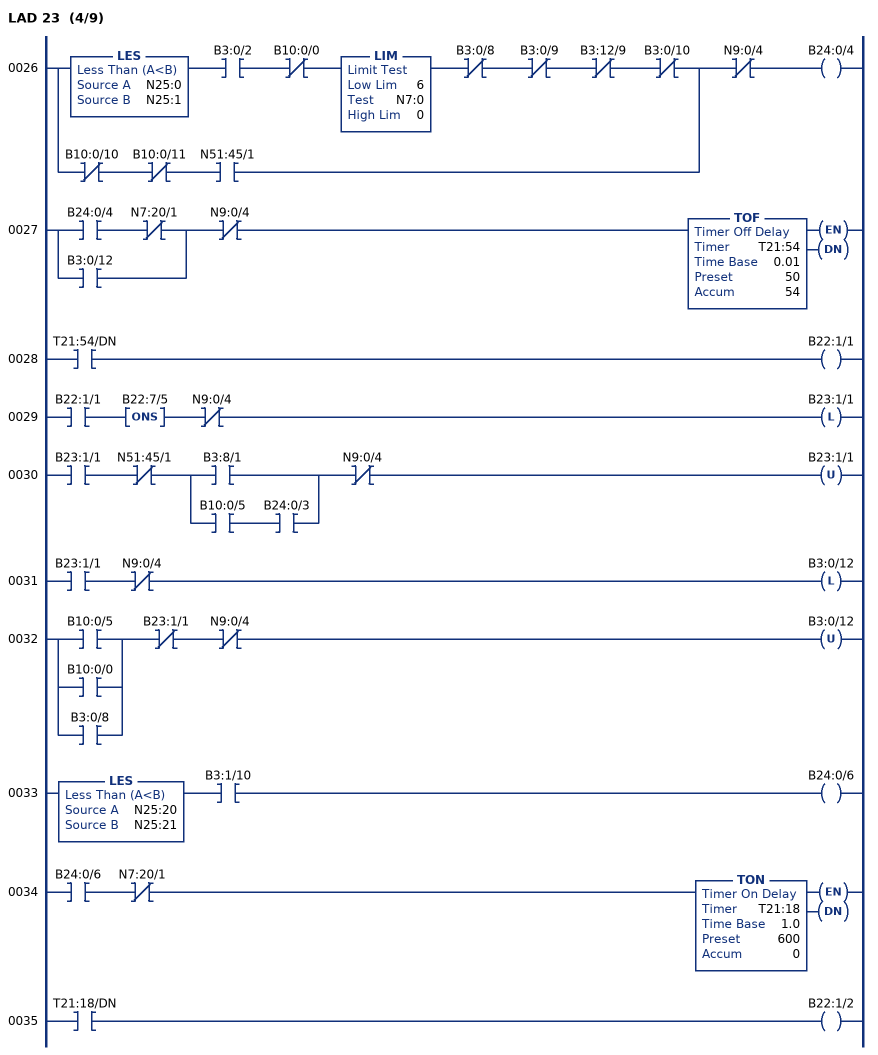
% Rung: 26 %
SOR BST LES N25:0 N25:1 XIC B3:0/2 XIO B10:0/0 LIM 6 N7:0 0 XIO B3:0/8 XIO B3:0/9 XIO B3:12/9 XIO B3:0/10 NXB XIO B10:0/10 XIO B10:0/11 XIC N51:45/1 BND XIO N9:0/4 OTE B24:0/4 EOR
% Rung: 27 %
SOR BST XIC B24:0/4 XIO N7:20/1 NXB XIC B3:0/12 BND XIO N9:0/4 TOF T21:54 0.01 50 54 EOR
% Rung: 28 %
SOR XIC T21:54/DN OTE B22:1/1 EOR
% Rung: 29 %
SOR XIC B22:1/1 OSR B22:7/5 XIO N9:0/4 OTL B23:1/1 EOR
% Rung: 30 %
SOR XIC B23:1/1 XIO N51:45/1 BST XIC B3:8/1 NXB XIC B10:0/5 XIC B24:0/3 BND XIO N9:0/4 OTU B23:1/1 EOR
% Rung: 31 %
SOR XIC B23:1/1 XIO N9:0/4 OTL B3:0/12 EOR
% Rung: 32 %
SOR BST XIC B10:0/5 NXB XIC B10:0/0 NXB XIC B3:0/8 BND XIO B23:1/1 XIO N9:0/4 OTU B3:0/12 EOR
% Rung: 33 %
SOR LES N25:20 N25:21 XIC B3:1/10 OTE B24:0/6 EOR
% Rung: 34 %
SOR XIC B24:0/6 XIO N7:20/1 TON T21:18 1.0 600 0 EOR
% Rung: 35 %
SOR XIC T21:18/DN OTE B22:1/2 EOR

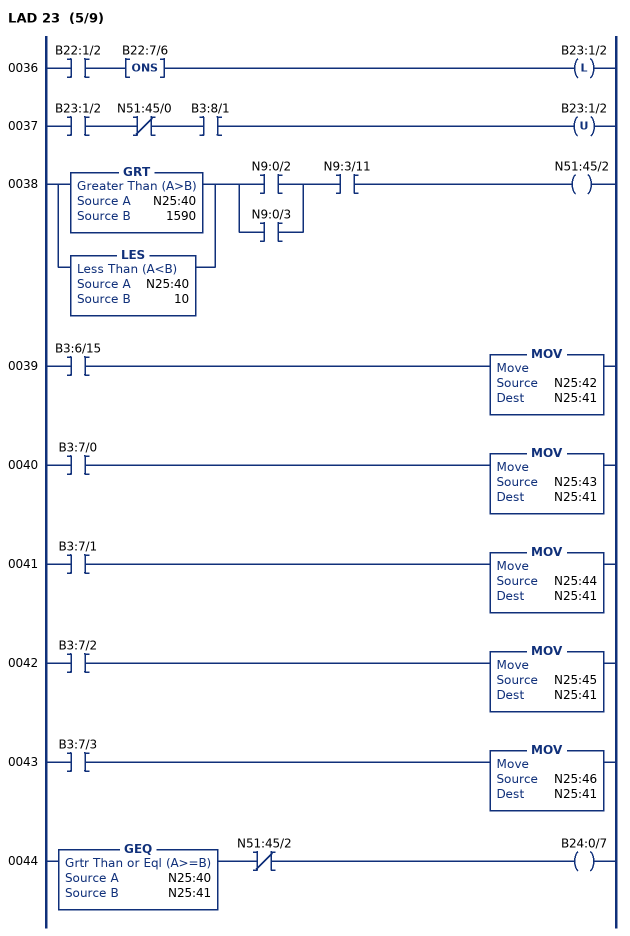
% Rung: 36 %
SOR XIC B22:1/2 OSR B22:7/6 OTL B23:1/2 EOR
% Rung: 37 %
SOR XIC B23:1/2 XIO N51:45/0 XIC B3:8/1 OTU B23:1/2 EOR
% Rung: 38 %
SOR BST GRT N25:40 1590 NXB LES N25:40 10 BND BST XIC N9:0/2 NXB XIC N9:0/3 BND XIC N9:3/11 OTE N51:45/2 EOR
% Rung: 39 %
SOR XIC B3:6/15 MOV N25:42 N25:41 EOR
% Rung: 40 %
SOR XIC B3:7/0 MOV N25:43 N25:41 EOR
% Rung: 41 %
SOR XIC B3:7/1 MOV N25:44 N25:41 EOR
% Rung: 42 %
SOR XIC B3:7/2 MOV N25:45 N25:41 EOR
% Rung: 43 %
SOR XIC B3:7/3 MOV N25:46 N25:41 EOR
% Rung: 44 %
SOR GEQ N25:40 N25:41 XIO N51:45/2 OTE B24:0/7 EOR

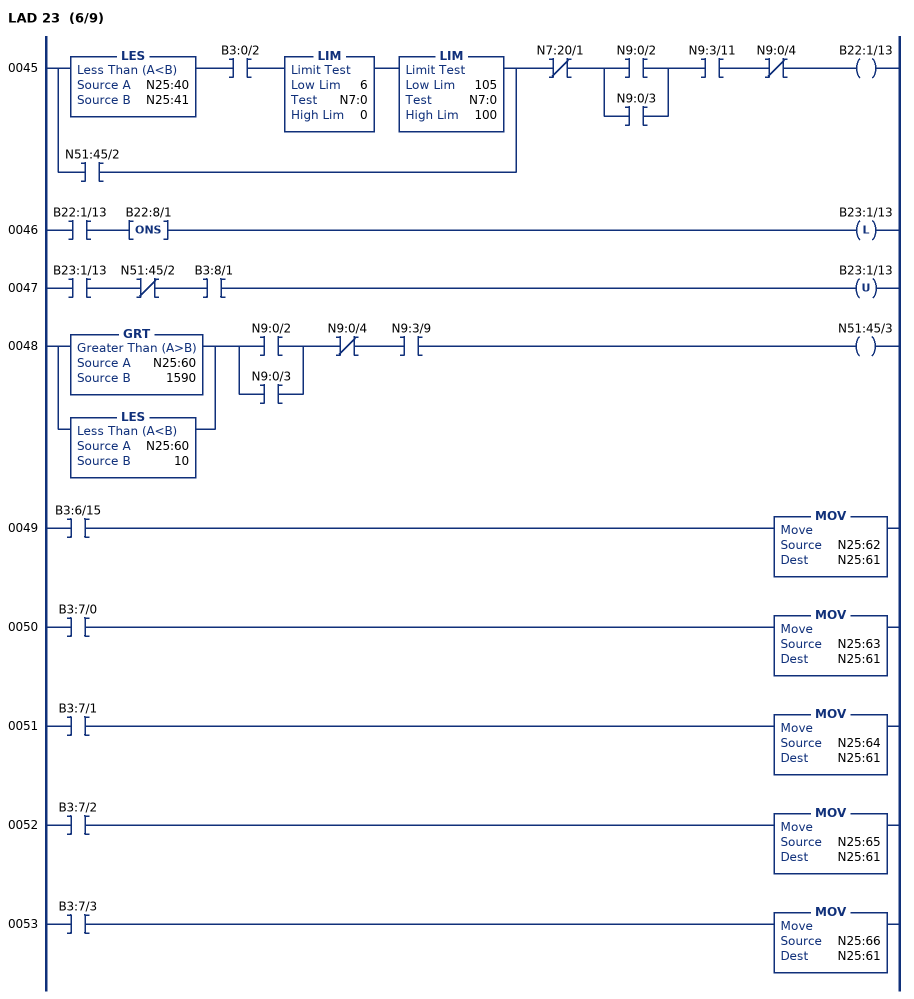
% Rung: 45 %
SOR BST LES N25:40 N25:41 XIC B3:0/2 LIM 6 N7:0 0 LIM 105 N7:0 100 NXB XIC N51:45/2 BND XIO N7:20/1 BST XIC N9:0/2 NXB XIC N9:0/3 BND XIC N9:3/11 XIO N9:0/4 OTE B22:1/13 EOR
% Rung: 46 %
SOR XIC B22:1/13 OSR B22:8/1 OTL B23:1/13 EOR
% Rung: 47 %
SOR XIC B23:1/13 XIO N51:45/2 XIC B3:8/1 OTU B23:1/13 EOR
% Rung: 48 %
SOR BST GRT N25:60 1590 NXB LES N25:60 10 BND BST XIC N9:0/2 NXB XIC N9:0/3 BND XIO N9:0/4 XIC N9:3/9 OTE N51:45/3 EOR
% Rung: 49 %
SOR XIC B3:6/15 MOV N25:62 N25:61 EOR
% Rung: 50 %
SOR XIC B3:7/0 MOV N25:63 N25:61 EOR
% Rung: 51 %
SOR XIC B3:7/1 MOV N25:64 N25:61 EOR
% Rung: 52 %
SOR XIC B3:7/2 MOV N25:65 N25:61 EOR
% Rung: 53 %
SOR XIC B3:7/3 MOV N25:66 N25:61 EOR

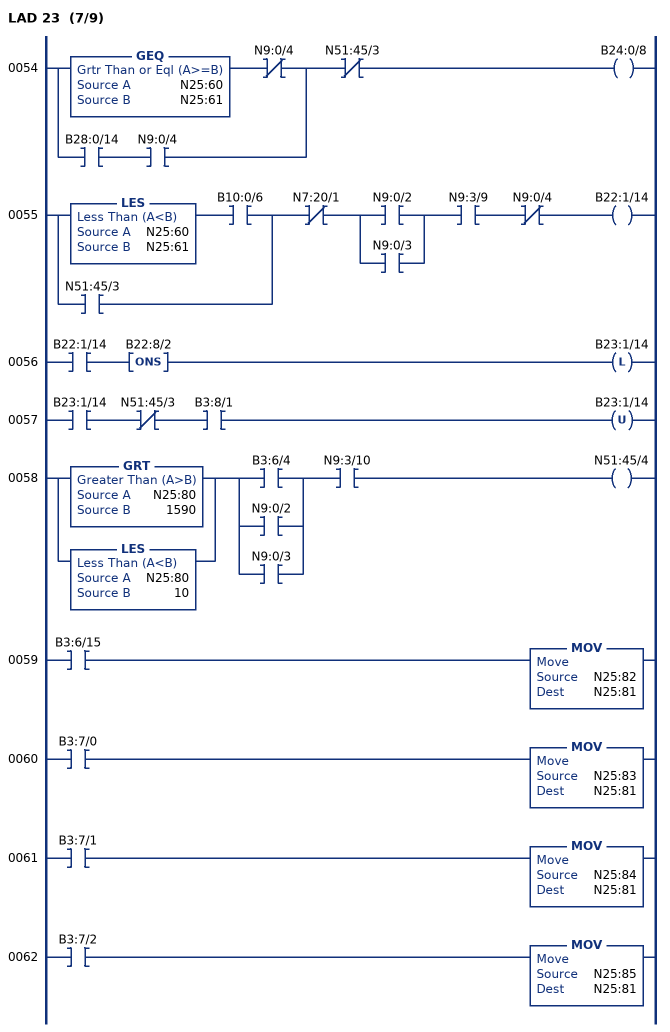
% Rung: 54 %
SOR BST GEQ N25:60 N25:61 XIO N9:0/4 NXB XIC B28:0/14 XIC N9:0/4 BND XIO N51:45/3 OTE B24:0/8 EOR
% Rung: 55 %
SOR BST LES N25:60 N25:61 XIC B10:0/6 NXB XIC N51:45/3 BND XIO N7:20/1 BST XIC N9:0/2 NXB XIC N9:0/3 BND XIC N9:3/9 XIO N9:0/4 OTE B22:1/14 EOR
% Rung: 56 %
SOR XIC B22:1/14 OSR B22:8/2 OTL B23:1/14 EOR
% Rung: 57 %
SOR XIC B23:1/14 XIO N51:45/3 XIC B3:8/1 OTU B23:1/14 EOR
% Rung: 58 %
SOR BST GRT N25:80 1590 NXB LES N25:80 10 BND BST XIC B3:6/4 NXB XIC N9:0/2 NXB XIC N9:0/3 BND XIC N9:3/10 OTE N51:45/4 EOR
% Rung: 59 %
SOR XIC B3:6/15 MOV N25:82 N25:81 EOR
% Rung: 60 %
SOR XIC B3:7/0 MOV N25:83 N25:81 EOR
% Rung: 61 %
SOR XIC B3:7/1 MOV N25:84 N25:81 EOR
% Rung: 62 %
SOR XIC B3:7/2 MOV N25:85 N25:81 EOR

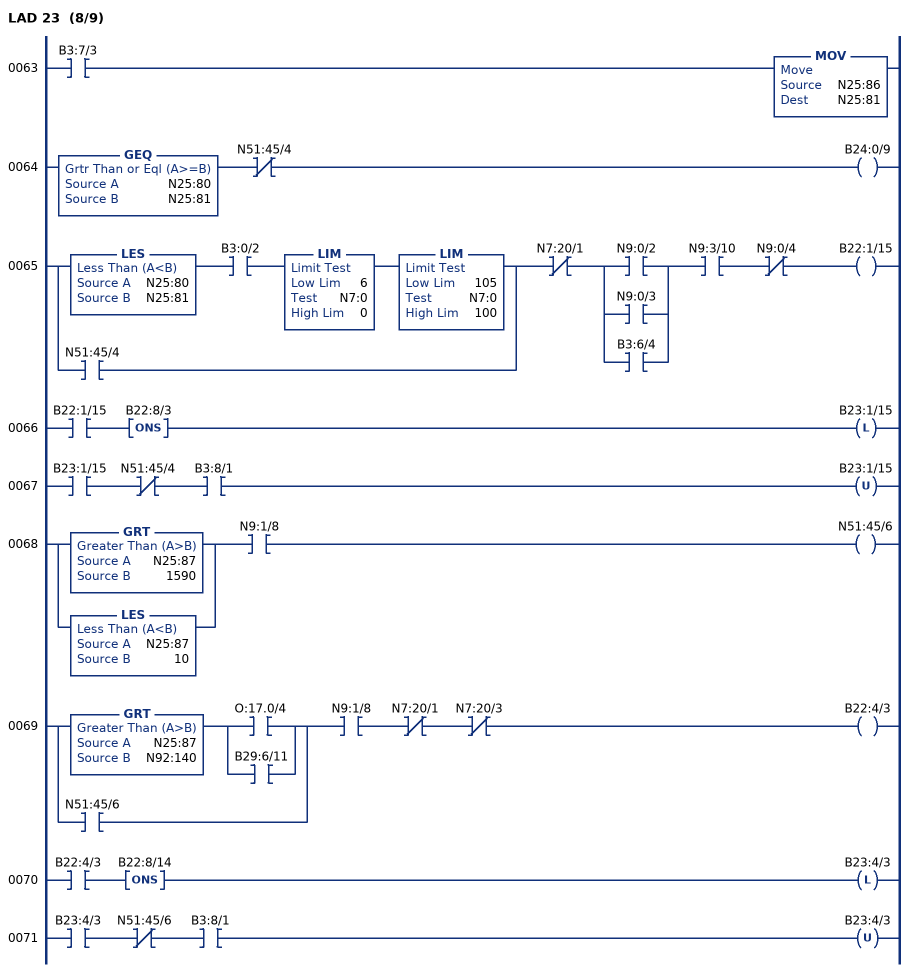
% Rung: 63 %
SOR XIC B3:7/3 MOV N25:86 N25:81 EOR
% Rung: 64 %
SOR GEQ N25:80 N25:81 XIO N51:45/4 OTE B24:0/9 EOR
% Rung: 65 %
SOR BST LES N25:80 N25:81 XIC B3:0/2 LIM 6 N7:0 0 LIM 105 N7:0 100 NXB XIC N51:45/4 BND XIO N7:20/1 BST XIC N9:0/2 NXB XIC N9:0/3 NXB XIC B3:6/4 BND XIC N9:3/10 XIO N9:0/4 OTE B22:1/15 EOR
% Rung: 66 %
SOR XIC B22:1/15 OSR B22:8/3 OTL B23:1/15 EOR
% Rung: 67 %
SOR XIC B23:1/15 XIO N51:45/4 XIC B3:8/1 OTU B23:1/15 EOR
% Rung: 68 %
SOR BST GRT N25:87 1590 NXB LES N25:87 10 BND XIC N9:1/8 OTE N51:45/6 EOR
% Rung: 69 %
SOR BST GRT N25:87 N92:140 BST XIC O:17.0/4 NXB XIC B29:6/11 BND NXB XIC N51:45/6 BND XIC N9:1/8 XIO N7:20/1 XIO N7:20/3 OTE B22:4/3 EOR
% Rung: 70 %
SOR XIC B22:4/3 OSR B22:8/14 OTL B23:4/3 EOR
% Rung: 71 %
SOR XIC B23:4/3 XIO N51:45/6 XIC B3:8/1 OTU B23:4/3 EOR

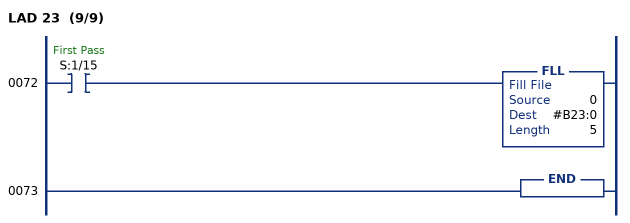
% Rung: 72 %
SOR XIC S:1/15 FLL 0 #B23:0 5 EOR
%   S:1/15  "First Pass" %
% Rung: 73 %
SOR END EOR

LADDER 24
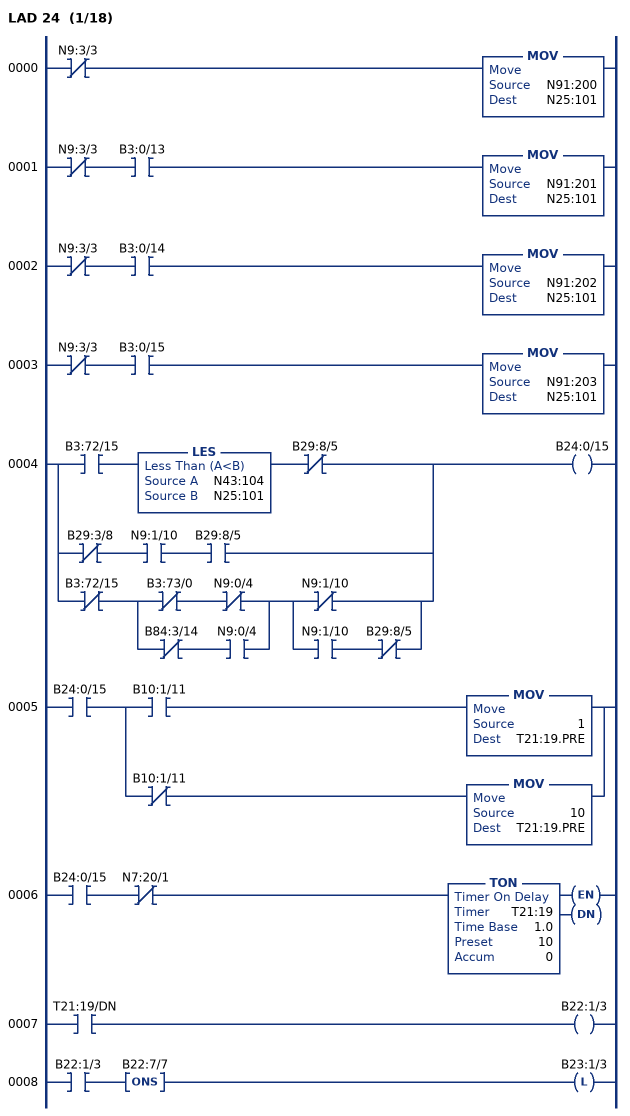
% Rung: 0 %
SOR XIO N9:3/3 MOV N91:200 N25:101 EOR
% Rung: 1 %
SOR XIO N9:3/3 XIC B3:0/13 MOV N91:201 N25:101 EOR
% Rung: 2 %
SOR XIO N9:3/3 XIC B3:0/14 MOV N91:202 N25:101 EOR
% Rung: 3 %
SOR XIO N9:3/3 XIC B3:0/15 MOV N91:203 N25:101 EOR
% Rung: 4 %
SOR BST XIC B3:72/15 LES N43:104 N25:101 XIO B29:8/5 NXB XIO B29:3/8 XIC N9:1/10 XIC B29:8/5 NXB XIO B3:72/15 BST XIO B3:73/0 XIO N9:0/4 NXB XIO B84:3/14 XIC N9:0/4 BND BST XIO N9:1/10 NXB XIC N9:1/10 XIO B29:8/5 BND BND OTE B24:0/15 EOR
% Rung: 5 %
SOR XIC B24:0/15 BST XIC B10:1/11 MOV 1 T21:19.PRE NXB XIO B10:1/11 MOV 10 T21:19.PRE BND EOR
% Rung: 6 %
SOR XIC B24:0/15 XIO N7:20/1 TON T21:19 1.0 10 0 EOR
% Rung: 7 %
SOR XIC T21:19/DN OTE B22:1/3 EOR
% Rung: 8 %
SOR XIC B22:1/3 OSR B22:7/7 OTL B23:1/3 EOR

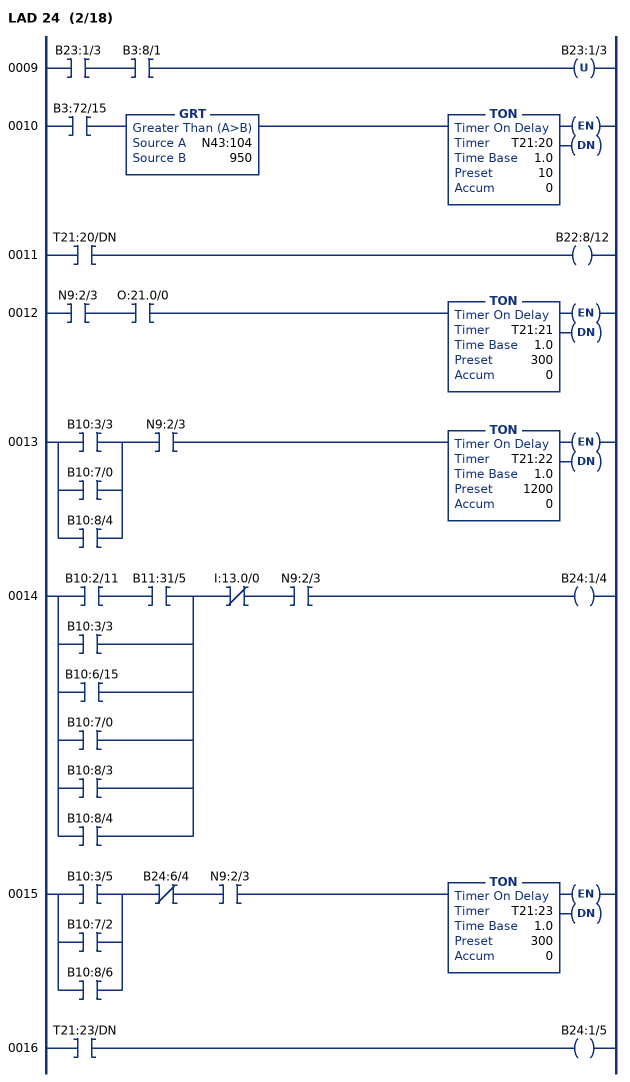
% Rung: 9 %
SOR XIC B23:1/3 XIC B3:8/1 OTU B23:1/3 EOR
% Rung: 10 %
SOR XIC B3:72/15 GRT N43:104 950 TON T21:20 1.0 10 0 EOR
% Rung: 11 %
SOR XIC T21:20/DN OTE B22:8/12 EOR
% Rung: 12 %
SOR XIC N9:2/3 XIC O:21.0/0 TON T21:21 1.0 300 0 EOR
% Rung: 13 %
SOR BST XIC B10:3/3 NXB XIC B10:7/0 NXB XIC B10:8/4 BND XIC N9:2/3 TON T21:22 1.0 1200 0 EOR
% Rung: 14 %
SOR BST XIC B10:2/11 XIC B11:31/5 NXB XIC B10:3/3 NXB XIC B10:6/15 NXB XIC B10:7/0 NXB XIC B10:8/3 NXB XIC B10:8/4 BND XIO I:13.0/0 XIC N9:2/3 OTE B24:1/4 EOR
% Rung: 15 %
SOR BST XIC B10:3/5 NXB XIC B10:7/2 NXB XIC B10:8/6 BND XIO B24:6/4 XIC N9:2/3 TON T21:23 1.0 300 0 EOR
% Rung: 16 %
SOR XIC T21:23/DN OTE B24:1/5 EOR

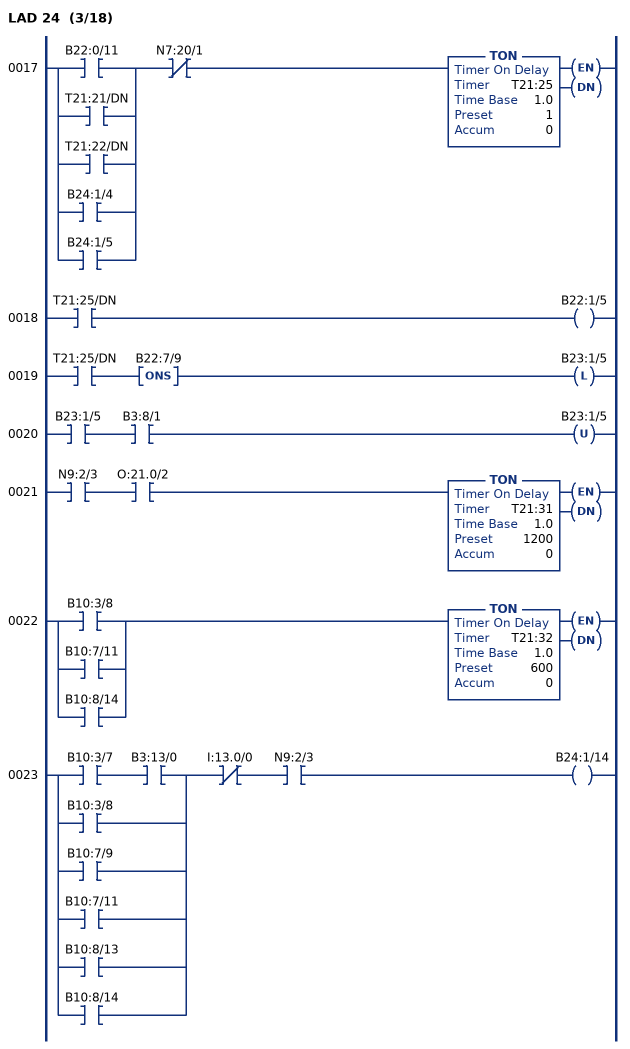
% Rung: 17 %
SOR BST XIC B22:0/11 NXB XIC T21:21/DN NXB XIC T21:22/DN NXB XIC B24:1/4 NXB XIC B24:1/5 BND XIO N7:20/1 TON T21:25 1.0 1 0 EOR
% Rung: 18 %
SOR XIC T21:25/DN OTE B22:1/5 EOR
% Rung: 19 %
SOR XIC T21:25/DN OSR B22:7/9 OTL B23:1/5 EOR
% Rung: 20 %
SOR XIC B23:1/5 XIC B3:8/1 OTU B23:1/5 EOR
% Rung: 21 %
SOR XIC N9:2/3 XIC O:21.0/2 TON T21:31 1.0 1200 0 EOR
% Rung: 22 %
SOR BST XIC B10:3/8 NXB XIC B10:7/11 NXB XIC B10:8/14 BND TON T21:32 1.0 600 0 EOR
% Rung: 23 %
SOR BST XIC B10:3/7 XIC B3:13/0 NXB XIC B10:3/8 NXB XIC B10:7/9 NXB XIC B10:7/11 NXB XIC B10:8/13 NXB XIC B10:8/14 BND XIO I:13.0/0 XIC N9:2/3 OTE B24:1/14 EOR

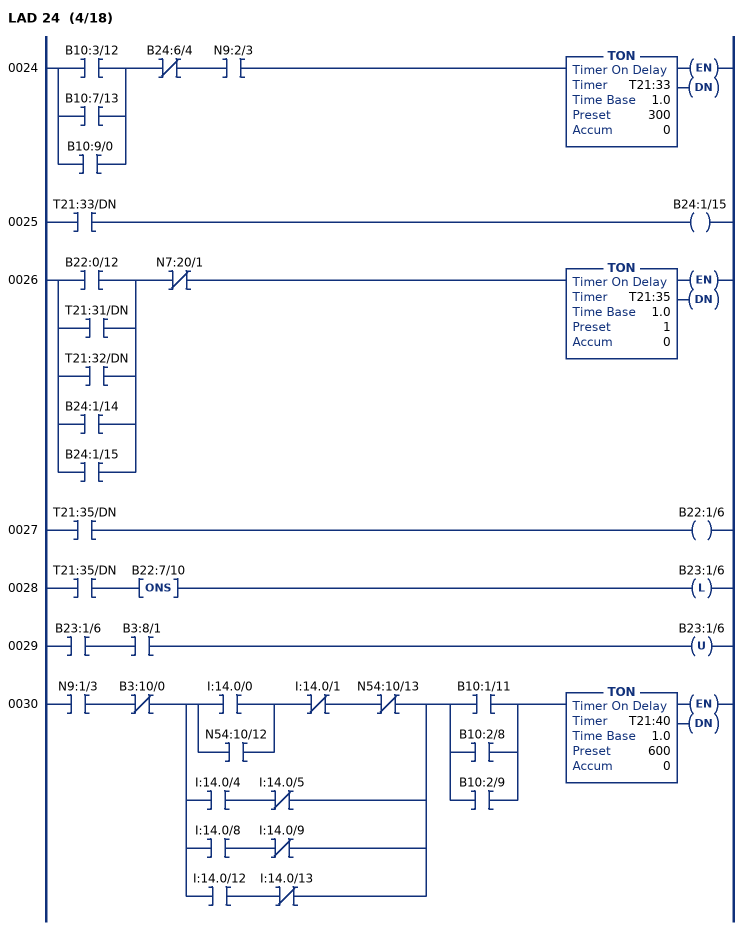
% Rung: 24 %
SOR BST XIC B10:3/12 NXB XIC B10:7/13 NXB XIC B10:9/0 BND XIO B24:6/4 XIC N9:2/3 TON T21:33 1.0 300 0 EOR
% Rung: 25 %
SOR XIC T21:33/DN OTE B24:1/15 EOR
% Rung: 26 %
SOR BST XIC B22:0/12 NXB XIC T21:31/DN NXB XIC T21:32/DN NXB XIC B24:1/14 NXB XIC B24:1/15 BND XIO N7:20/1 TON T21:35 1.0 1 0 EOR
% Rung: 27 %
SOR XIC T21:35/DN OTE B22:1/6 EOR
% Rung: 28 %
SOR XIC T21:35/DN OSR B22:7/10 OTL B23:1/6 EOR
% Rung: 29 %
SOR XIC B23:1/6 XIC B3:8/1 OTU B23:1/6 EOR
% Rung: 30 %
SOR XIC N9:1/3 XIO B3:10/0 BST BST XIC I:14.0/0 NXB XIC N54:10/12 BND XIO I:14.0/1 XIO N54:10/13 NXB XIC I:14.0/4 XIO I:14.0/5 NXB XIC I:14.0/8 XIO I:14.0/9 NXB XIC I:14.0/12 XIO I:14.0/13 BND BST XIC B10:1/11 NXB XIC B10:2/8 NXB XIC B10:2/9 BND TON T21:40 1.0 600 0 EOR

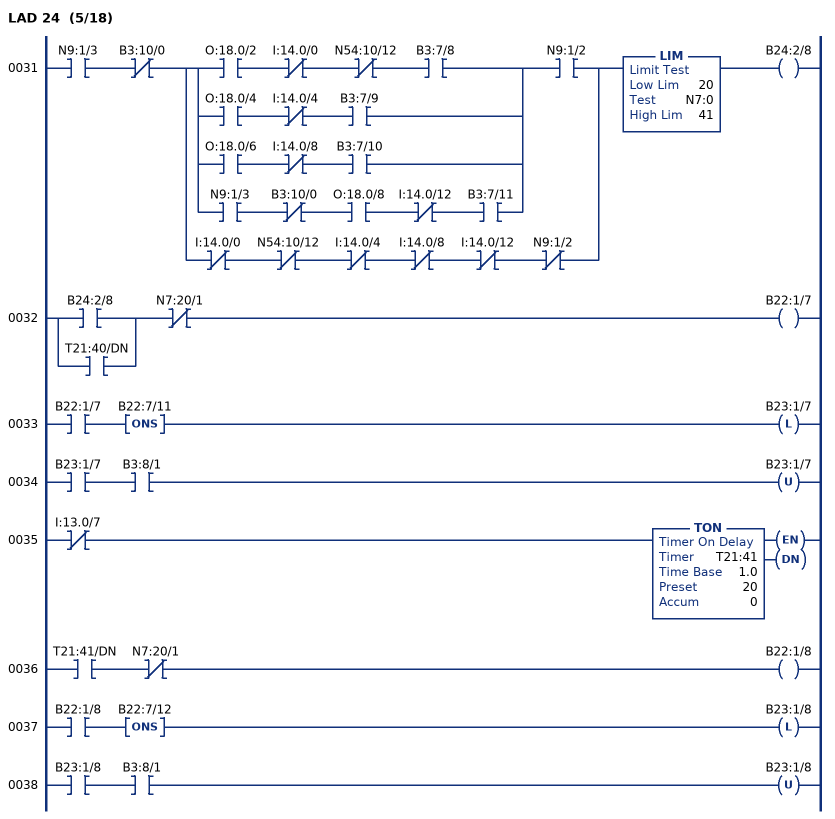
% Rung: 31 %
SOR XIC N9:1/3 XIO B3:10/0 BST BST XIC O:18.0/2 XIO I:14.0/0 XIO N54:10/12 XIC B3:7/8 NXB XIC O:18.0/4 XIO I:14.0/4 XIC B3:7/9 NXB XIC O:18.0/6 XIO I:14.0/8 XIC B3:7/10 NXB XIC N9:1/3 XIO B3:10/0 XIC O:18.0/8 XIO I:14.0/12 XIC B3:7/11 BND XIC N9:1/2 NXB XIO I:14.0/0 XIO N54:10/12 XIO I:14.0/4 XIO I:14.0/8 XIO I:14.0/12 XIO N9:1/2 BND LIM 20 N7:0 41 OTE B24:2/8 EOR
% Rung: 32 %
SOR BST XIC B24:2/8 NXB XIC T21:40/DN BND XIO N7:20/1 OTE B22:1/7 EOR
% Rung: 33 %
SOR XIC B22:1/7 OSR B22:7/11 OTL B23:1/7 EOR
% Rung: 34 %
SOR XIC B23:1/7 XIC B3:8/1 OTU B23:1/7 EOR
% Rung: 35 %
SOR XIO I:13.0/7 TON T21:41 1.0 20 0 EOR
% Rung: 36 %
SOR XIC T21:41/DN XIO N7:20/1 OTE B22:1/8 EOR
% Rung: 37 %
SOR XIC B22:1/8 OSR B22:7/12 OTL B23:1/8 EOR
% Rung: 38 %
SOR XIC B23:1/8 XIC B3:8/1 OTU B23:1/8 EOR

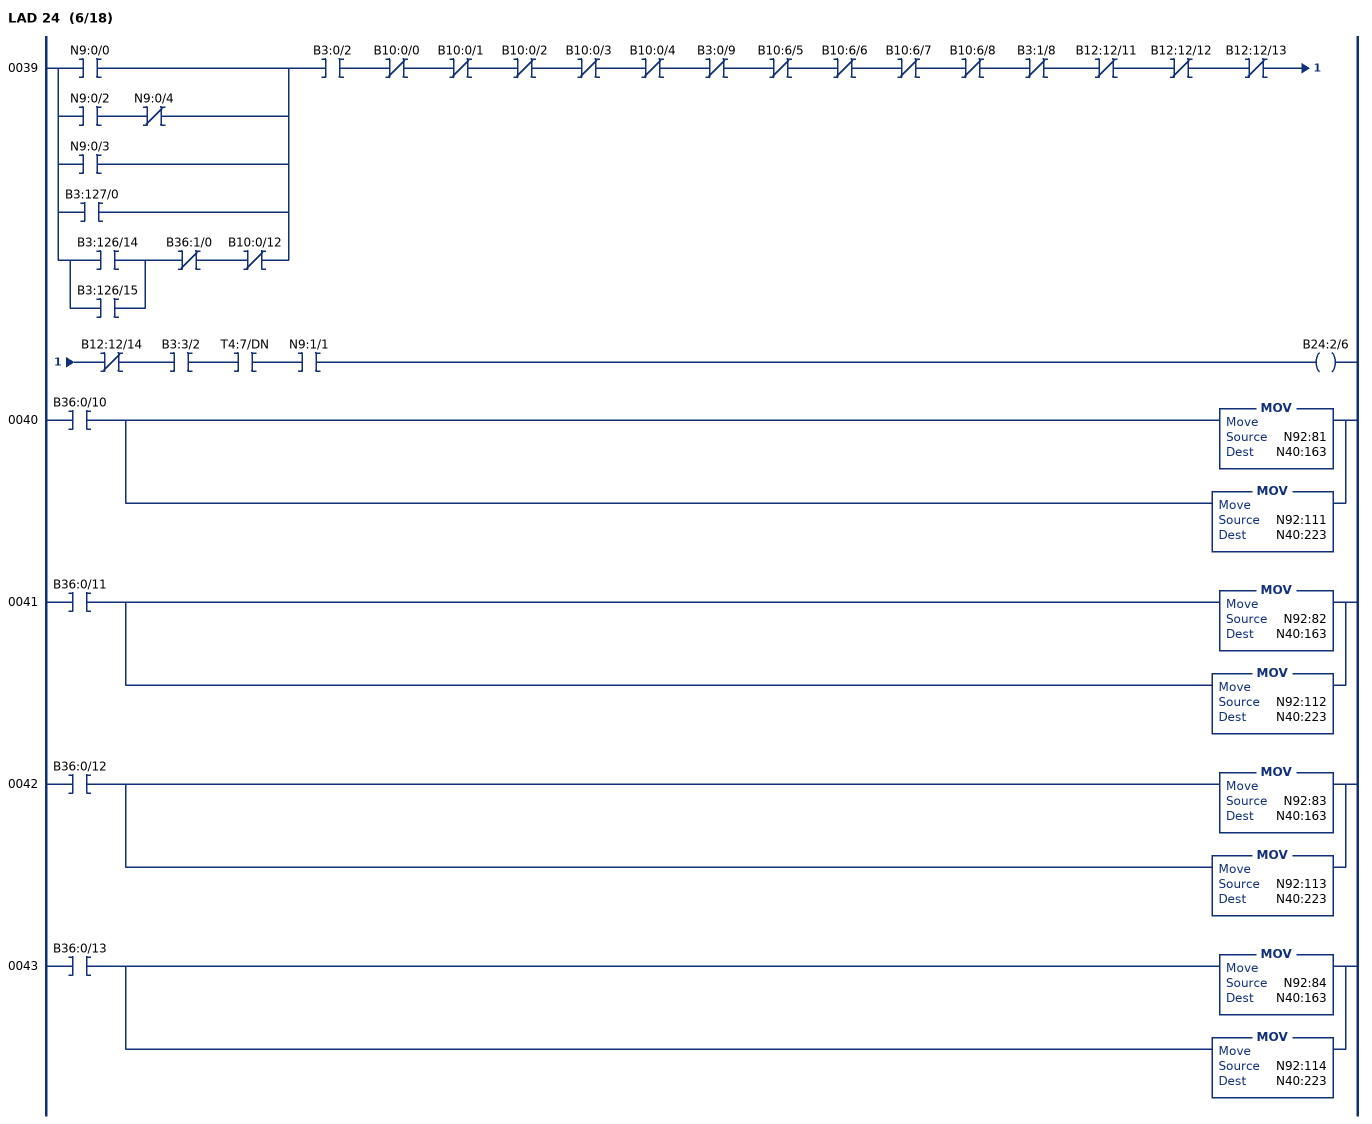
% Rung: 39 %
SOR BST XIC N9:0/0 NXB XIC N9:0/2 XIO N9:0/4 NXB XIC N9:0/3 NXB XIC B3:127/0 NXB BST XIC B3:126/14 NXB XIC B3:126/15 BND XIO B36:1/0 XIO B10:0/12 BND XIC B3:0/2 XIO B10:0/0 XIO B10:0/1 XIO B10:0/2 XIO B10:0/3 XIO B10:0/4 XIO B3:0/9 XIO B10:6/5 XIO B10:6/6 XIO B10:6/7 XIO B10:6/8 XIO B3:1/8 XIO B12:12/11 XIO B12:12/12 XIO B12:12/13 XIO B12:12/14 XIC B3:3/2 XIC T4:7/DN XIC N9:1/1 OTE B24:2/6 EOR
% Rung: 40 %
SOR XIC B36:0/10 BST MOV N92:81 N40:163 NXB MOV N92:111 N40:223 BND EOR
% Rung: 41 %
SOR XIC B36:0/11 BST MOV N92:82 N40:163 NXB MOV N92:112 N40:223 BND EOR
% Rung: 42 %
SOR XIC B36:0/12 BST MOV N92:83 N40:163 NXB MOV N92:113 N40:223 BND EOR
% Rung: 43 %
SOR XIC B36:0/13 BST MOV N92:84 N40:163 NXB MOV N92:114 N40:223 BND EOR

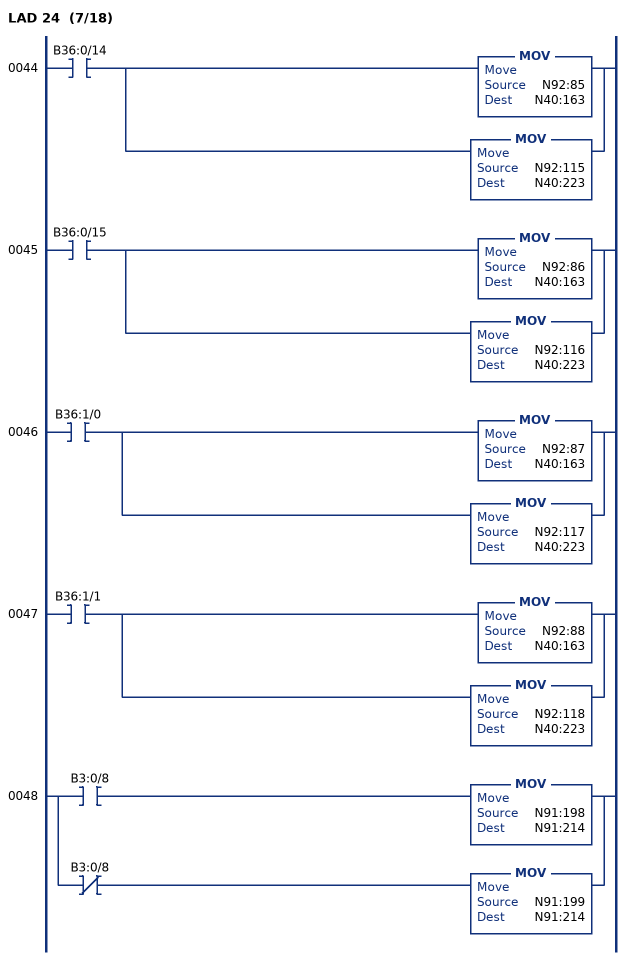
% Rung: 44 %
SOR XIC B36:0/14 BST MOV N92:85 N40:163 NXB MOV N92:115 N40:223 BND EOR
% Rung: 45 %
SOR XIC B36:0/15 BST MOV N92:86 N40:163 NXB MOV N92:116 N40:223 BND EOR
% Rung: 46 %
SOR XIC B36:1/0 BST MOV N92:87 N40:163 NXB MOV N92:117 N40:223 BND EOR
% Rung: 47 %
SOR XIC B36:1/1 BST MOV N92:88 N40:163 NXB MOV N92:118 N40:223 BND EOR
% Rung: 48 %
SOR BST XIC B3:0/8 MOV N91:198 N91:214 NXB XIO B3:0/8 MOV N91:199 N91:214 BND EOR

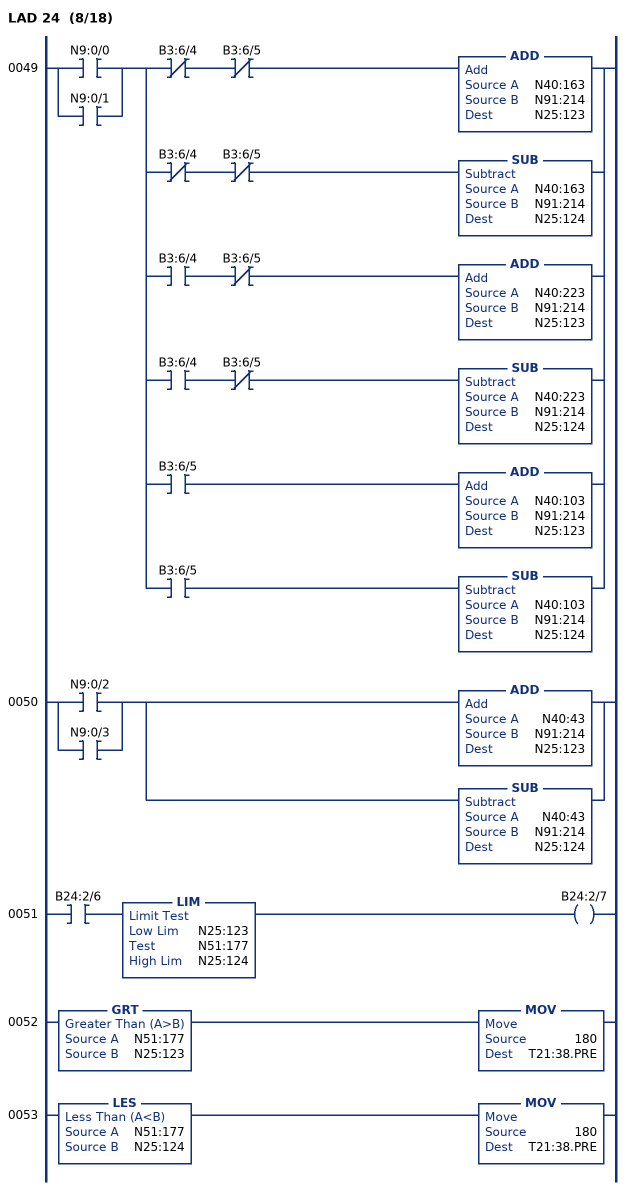
% Rung: 49 %
SOR BST XIC N9:0/0 NXB XIC N9:0/1 BND BST XIO B3:6/4 XIO B3:6/5 ADD N40:163 N91:214 N25:123 NXB XIO B3:6/4 XIO B3:6/5 SUB N40:163 N91:214 N25:124 NXB XIC B3:6/4 XIO B3:6/5 ADD N40:223 N91:214 N25:123 NXB XIC B3:6/4 XIO B3:6/5 SUB N40:223 N91:214 N25:124 NXB XIC B3:6/5 ADD N40:103 N91:214 N25:123 NXB XIC B3:6/5 SUB N40:103 N91:214 N25:124 BND EOR
% Rung: 50 %
SOR BST XIC N9:0/2 NXB XIC N9:0/3 BND BST ADD N40:43 N91:214 N25:123 NXB SUB N40:43 N91:214 N25:124 BND EOR
% Rung: 51 %
SOR XIC B24:2/6 LIM N25:123 N51:177 N25:124 OTE B24:2/7 EOR
% Rung: 52 %
SOR GRT N51:177 N25:123 MOV 180 T21:38.PRE EOR
% Rung: 53 %
SOR LES N51:177 N25:124 MOV 180 T21:38.PRE EOR

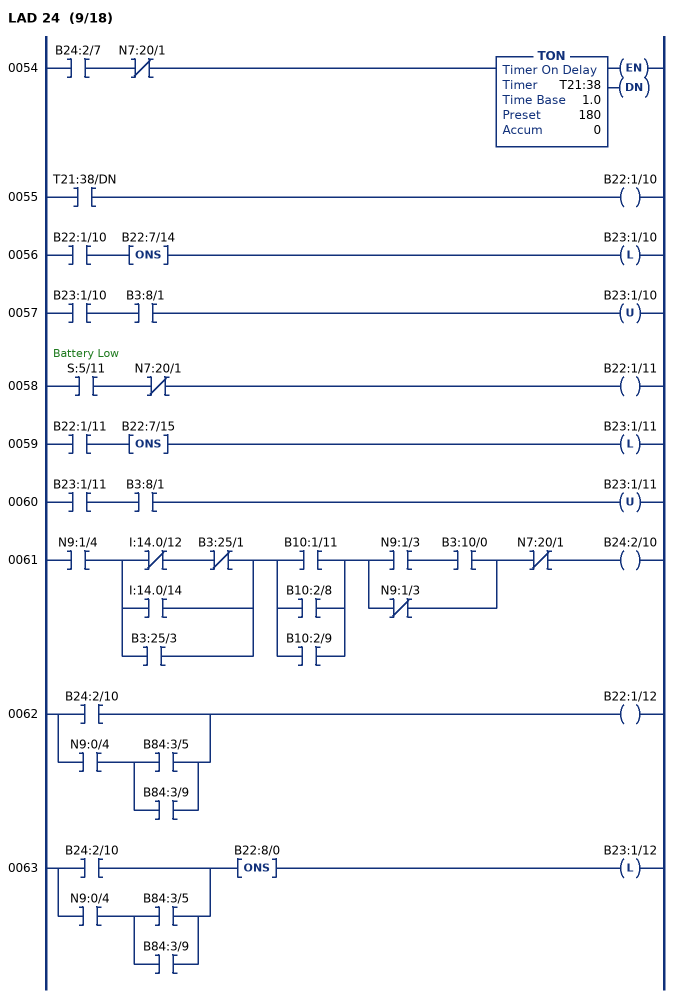
% Rung: 54 %
SOR XIC B24:2/7 XIO N7:20/1 TON T21:38 1.0 180 0 EOR
% Rung: 55 %
SOR XIC T21:38/DN OTE B22:1/10 EOR
% Rung: 56 %
SOR XIC B22:1/10 OSR B22:7/14 OTL B23:1/10 EOR
% Rung: 57 %
SOR XIC B23:1/10 XIC B3:8/1 OTU B23:1/10 EOR
% Rung: 58 %
SOR XIC S:5/11 XIO N7:20/1 OTE B22:1/11 EOR
%   S:5/11  "Battery Low" %
% Rung: 59 %
SOR XIC B22:1/11 OSR B22:7/15 OTL B23:1/11 EOR
% Rung: 60 %
SOR XIC B23:1/11 XIC B3:8/1 OTU B23:1/11 EOR
% Rung: 61 %
SOR XIC N9:1/4 BST XIO I:14.0/12 XIO B3:25/1 NXB XIC I:14.0/14 NXB XIC B3:25/3 BND BST XIC B10:1/11 NXB XIC B10:2/8 NXB XIC B10:2/9 BND BST XIC N9:1/3 XIC B3:10/0 NXB XIO N9:1/3 BND XIO N7:20/1 OTE B24:2/10 EOR
% Rung: 62 %
SOR BST XIC B24:2/10 NXB XIC N9:0/4 BST XIC B84:3/5 NXB XIC B84:3/9 BND BND OTE B22:1/12 EOR
% Rung: 63 %
SOR BST XIC B24:2/10 NXB XIC N9:0/4 BST XIC B84:3/5 NXB XIC B84:3/9 BND BND OSR B22:8/0 OTL B23:1/12 EOR

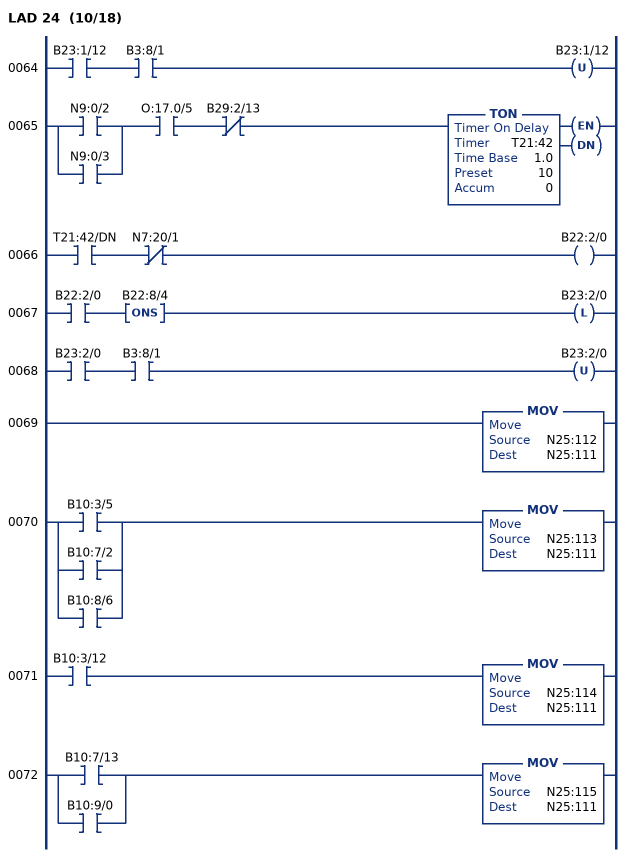
% Rung: 64 %
SOR XIC B23:1/12 XIC B3:8/1 OTU B23:1/12 EOR
% Rung: 65 %
SOR BST XIC N9:0/2 NXB XIC N9:0/3 BND XIC O:17.0/5 XIO B29:2/13 TON T21:42 1.0 10 0 EOR
% Rung: 66 %
SOR XIC T21:42/DN XIO N7:20/1 OTE B22:2/0 EOR
% Rung: 67 %
SOR XIC B22:2/0 OSR B22:8/4 OTL B23:2/0 EOR
% Rung: 68 %
SOR XIC B23:2/0 XIC B3:8/1 OTU B23:2/0 EOR
% Rung: 69 %
SOR MOV N25:112 N25:111 EOR
% Rung: 70 %
SOR BST XIC B10:3/5 NXB XIC B10:7/2 NXB XIC B10:8/6 BND MOV N25:113 N25:111 EOR
% Rung: 71 %
SOR XIC B10:3/12 MOV N25:114 N25:111 EOR
% Rung: 72 %
SOR BST XIC B10:7/13 NXB XIC B10:9/0 BND MOV N25:115 N25:111 EOR

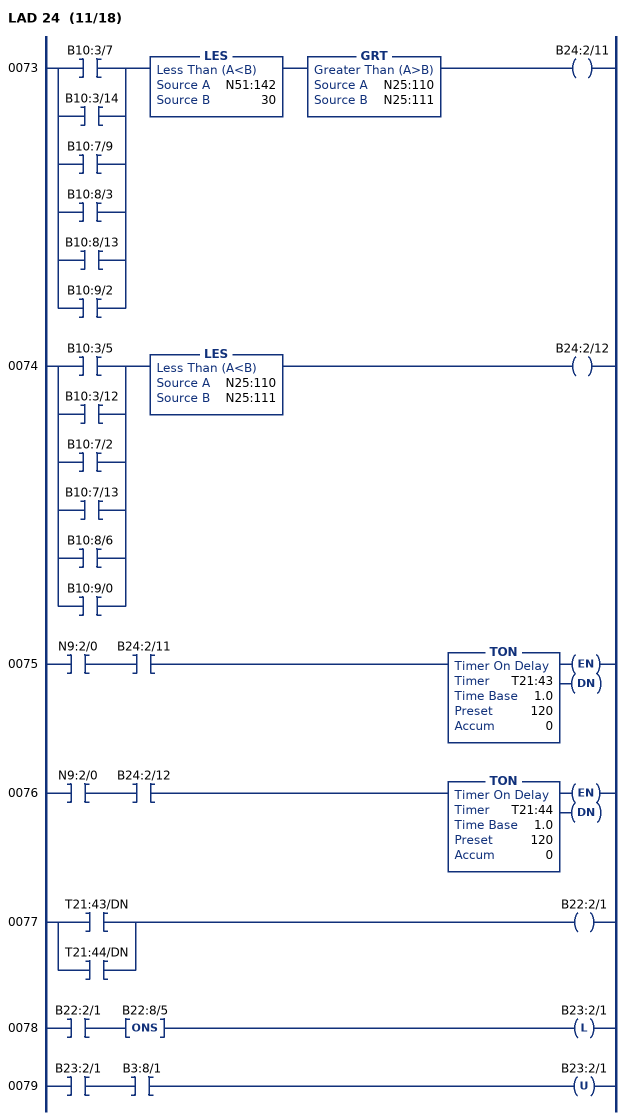
% Rung: 73 %
SOR BST XIC B10:3/7 NXB XIC B10:3/14 NXB XIC B10:7/9 NXB XIC B10:8/3 NXB XIC B10:8/13 NXB XIC B10:9/2 BND LES N51:142 30 GRT N25:110 N25:111 OTE B24:2/11 EOR
% Rung: 74 %
SOR BST XIC B10:3/5 NXB XIC B10:3/12 NXB XIC B10:7/2 NXB XIC B10:7/13 NXB XIC B10:8/6 NXB XIC B10:9/0 BND LES N25:110 N25:111 OTE B24:2/12 EOR
% Rung: 75 %
SOR XIC N9:2/0 XIC B24:2/11 TON T21:43 1.0 120 0 EOR
% Rung: 76 %
SOR XIC N9:2/0 XIC B24:2/12 TON T21:44 1.0 120 0 EOR
% Rung: 77 %
SOR BST XIC T21:43/DN NXB XIC T21:44/DN BND OTE B22:2/1 EOR
% Rung: 78 %
SOR XIC B22:2/1 OSR B22:8/5 OTL B23:2/1 EOR
% Rung: 79 %
SOR XIC B23:2/1 XIC B3:8/1 OTU B23:2/1 EOR

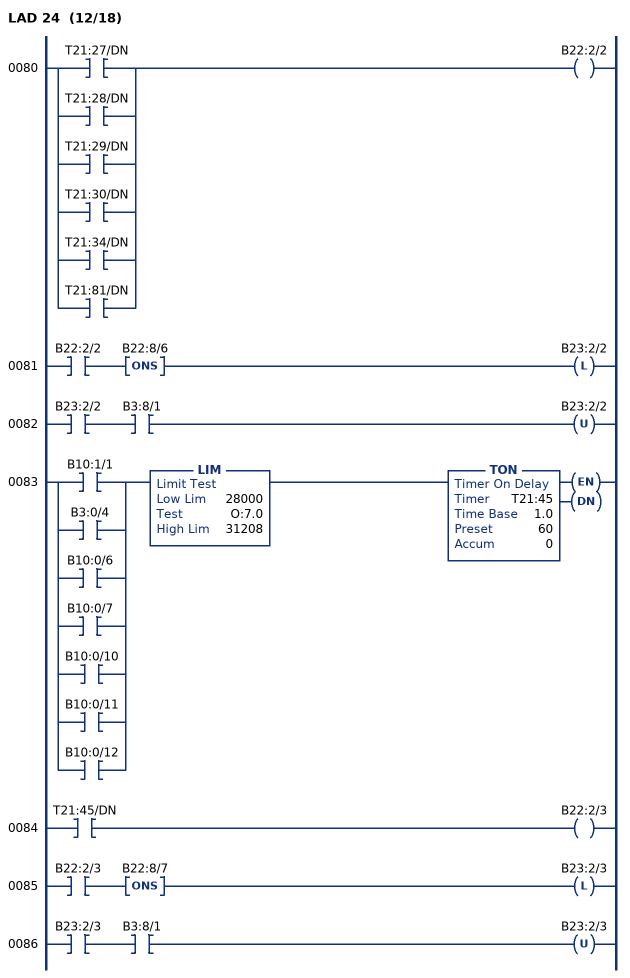
% Rung: 80 %
SOR BST XIC T21:27/DN NXB XIC T21:28/DN NXB XIC T21:29/DN NXB XIC T21:30/DN NXB XIC T21:34/DN NXB XIC T21:81/DN BND OTE B22:2/2 EOR
% Rung: 81 %
SOR XIC B22:2/2 OSR B22:8/6 OTL B23:2/2 EOR
% Rung: 82 %
SOR XIC B23:2/2 XIC B3:8/1 OTU B23:2/2 EOR
% Rung: 83 %
SOR BST XIC B10:1/1 NXB XIC B3:0/4 NXB XIC B10:0/6 NXB XIC B10:0/7 NXB XIC B10:0/10 NXB XIC B10:0/11 NXB XIC B10:0/12 BND LIM 28000 O:7.0 31208 TON T21:45 1.0 60 0 EOR
% Rung: 84 %
SOR XIC T21:45/DN OTE B22:2/3 EOR
% Rung: 85 %
SOR XIC B22:2/3 OSR B22:8/7 OTL B23:2/3 EOR
% Rung: 86 %
SOR XIC B23:2/3 XIC B3:8/1 OTU B23:2/3 EOR

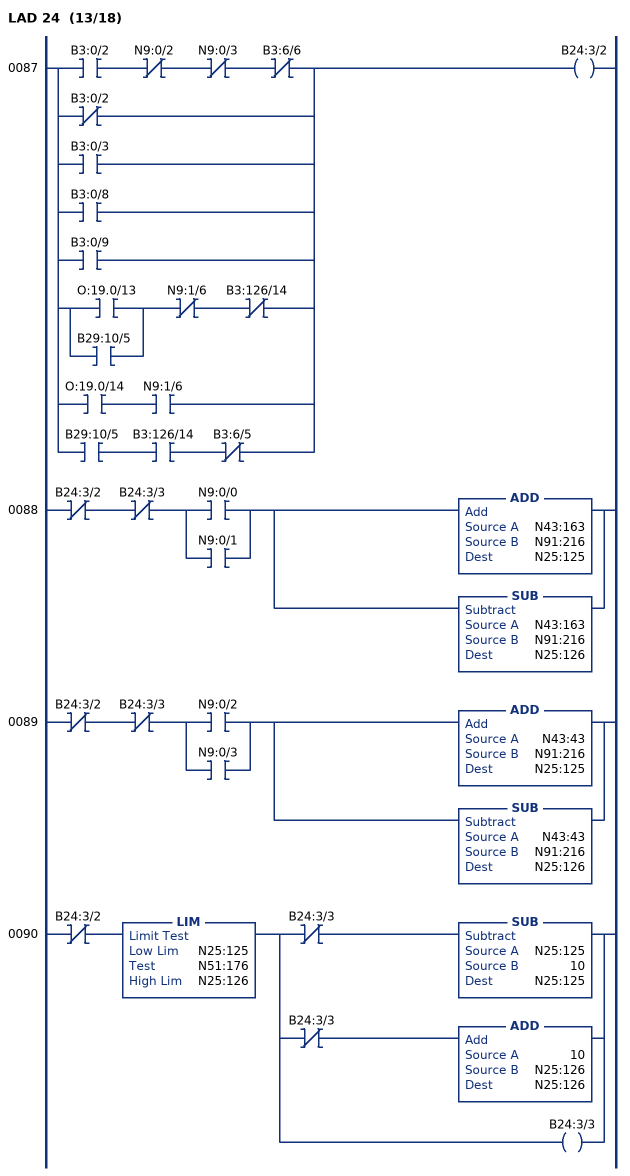
% Rung: 87 %
SOR BST XIC B3:0/2 XIO N9:0/2 XIO N9:0/3 XIO B3:6/6 NXB XIO B3:0/2 NXB XIC B3:0/3 NXB XIC B3:0/8 NXB XIC B3:0/9 NXB BST XIC O:19.0/13 NXB XIC B29:10/5 BND XIO N9:1/6 XIO B3:126/14 NXB XIC O:19.0/14 XIC N9:1/6 NXB XIC B29:10/5 XIC B3:126/14 XIO B3:6/5 BND OTE B24:3/2 EOR
% Rung: 88 %
SOR XIO B24:3/2 XIO B24:3/3 BST XIC N9:0/0 NXB XIC N9:0/1 BND BST ADD N43:163 N91:216 N25:125 NXB SUB N43:163 N91:216 N25:126 BND EOR
% Rung: 89 %
SOR XIO B24:3/2 XIO B24:3/3 BST XIC N9:0/2 NXB XIC N9:0/3 BND BST ADD N43:43 N91:216 N25:125 NXB SUB N43:43 N91:216 N25:126 BND EOR
% Rung: 90 %
SOR XIO B24:3/2 LIM N25:125 N51:176 N25:126 BST XIO B24:3/3 SUB N25:125 10 N25:125 NXB XIO B24:3/3 ADD 10 N25:126 N25:126 NXB OTE B24:3/3 BND EOR

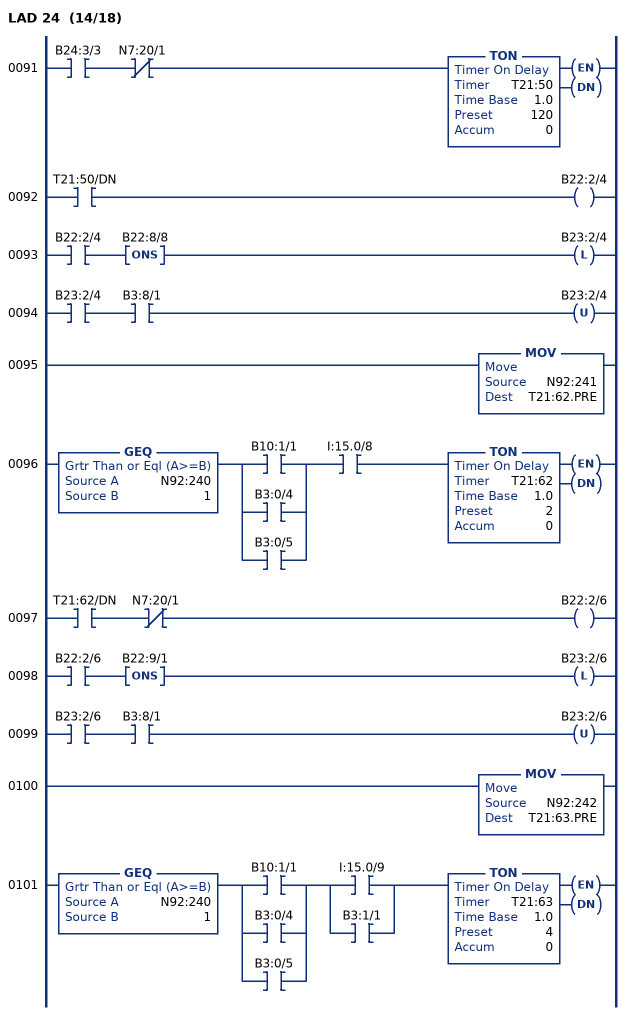
% Rung: 91 %
SOR XIC B24:3/3 XIO N7:20/1 TON T21:50 1.0 120 0 EOR
% Rung: 92 %
SOR XIC T21:50/DN OTE B22:2/4 EOR
% Rung: 93 %
SOR XIC B22:2/4 OSR B22:8/8 OTL B23:2/4 EOR
% Rung: 94 %
SOR XIC B23:2/4 XIC B3:8/1 OTU B23:2/4 EOR
% Rung: 95 %
SOR MOV N92:241 T21:62.PRE EOR
% Rung: 96 %
SOR GEQ N92:240 1 BST XIC B10:1/1 NXB XIC B3:0/4 NXB XIC B3:0/5 BND XIC I:15.0/8 TON T21:62 1.0 2 0 EOR
% Rung: 97 %
SOR XIC T21:62/DN XIO N7:20/1 OTE B22:2/6 EOR
% Rung: 98 %
SOR XIC B22:2/6 OSR B22:9/1 OTL B23:2/6 EOR
% Rung: 99 %
SOR XIC B23:2/6 XIC B3:8/1 OTU B23:2/6 EOR
% Rung: 100 %
SOR MOV N92:242 T21:63.PRE EOR
% Rung: 101 %
SOR GEQ N92:240 1 BST XIC B10:1/1 NXB XIC B3:0/4 NXB XIC B3:0/5 BND BST XIC I:15.0/9 NXB XIC B3:1/1 BND TON T21:63 1.0 4 0 EOR

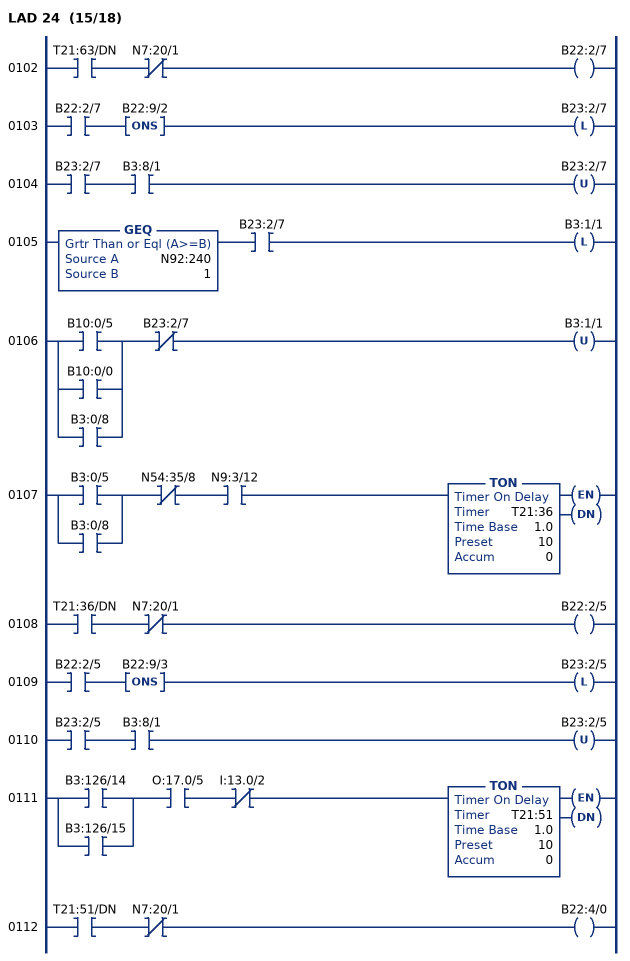
% Rung: 102 %
SOR XIC T21:63/DN XIO N7:20/1 OTE B22:2/7 EOR
% Rung: 103 %
SOR XIC B22:2/7 OSR B22:9/2 OTL B23:2/7 EOR
% Rung: 104 %
SOR XIC B23:2/7 XIC B3:8/1 OTU B23:2/7 EOR
% Rung: 105 %
SOR GEQ N92:240 1 XIC B23:2/7 OTL B3:1/1 EOR
% Rung: 106 %
SOR BST XIC B10:0/5 NXB XIC B10:0/0 NXB XIC B3:0/8 BND XIO B23:2/7 OTU B3:1/1 EOR
% Rung: 107 %
SOR BST XIC B3:0/5 NXB XIC B3:0/8 BND XIO N54:35/8 XIC N9:3/12 TON T21:36 1.0 10 0 EOR
% Rung: 108 %
SOR XIC T21:36/DN XIO N7:20/1 OTE B22:2/5 EOR
% Rung: 109 %
SOR XIC B22:2/5 OSR B22:9/3 OTL B23:2/5 EOR
% Rung: 110 %
SOR XIC B23:2/5 XIC B3:8/1 OTU B23:2/5 EOR
% Rung: 111 %
SOR BST XIC B3:126/14 NXB XIC B3:126/15 BND XIC O:17.0/5 XIO I:13.0/2 TON T21:51 1.0 10 0 EOR
% Rung: 112 %
SOR XIC T21:51/DN XIO N7:20/1 OTE B22:4/0 EOR

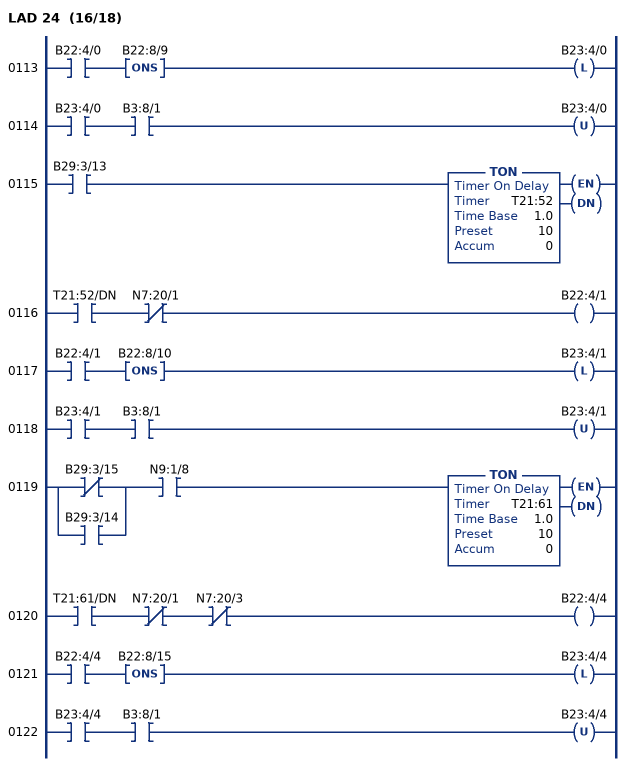
% Rung: 113 %
SOR XIC B22:4/0 OSR B22:8/9 OTL B23:4/0 EOR
% Rung: 114 %
SOR XIC B23:4/0 XIC B3:8/1 OTU B23:4/0 EOR
% Rung: 115 %
SOR XIC B29:3/13 TON T21:52 1.0 10 0 EOR
% Rung: 116 %
SOR XIC T21:52/DN XIO N7:20/1 OTE B22:4/1 EOR
% Rung: 117 %
SOR XIC B22:4/1 OSR B22:8/10 OTL B23:4/1 EOR
% Rung: 118 %
SOR XIC B23:4/1 XIC B3:8/1 OTU B23:4/1 EOR
% Rung: 119 %
SOR BST XIO B29:3/15 NXB XIC B29:3/14 BND XIC N9:1/8 TON T21:61 1.0 10 0 EOR
% Rung: 120 %
SOR XIC T21:61/DN XIO N7:20/1 XIO N7:20/3 OTE B22:4/4 EOR
% Rung: 121 %
SOR XIC B22:4/4 OSR B22:8/15 OTL B23:4/4 EOR
% Rung: 122 %
SOR XIC B23:4/4 XIC B3:8/1 OTU B23:4/4 EOR

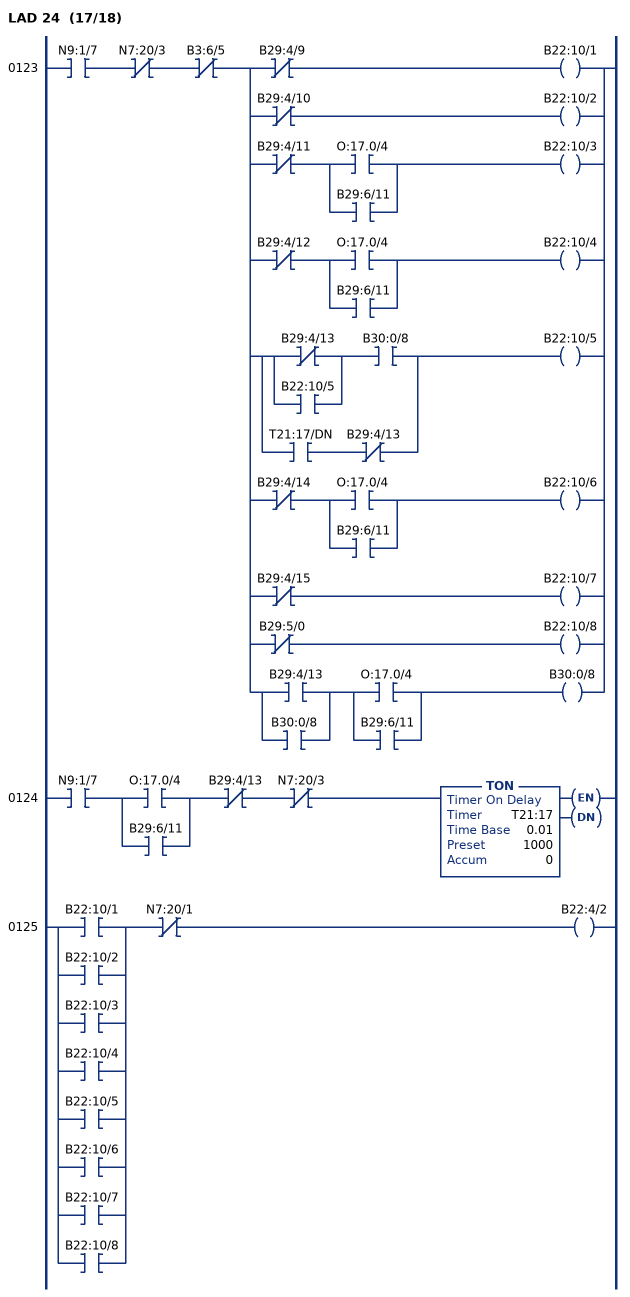
% Rung: 123 %
SOR XIC N9:1/7 XIO N7:20/3 XIO B3:6/5 BST XIO B29:4/9 OTE B22:10/1 NXB XIO B29:4/10 OTE B22:10/2 NXB XIO B29:4/11 BST XIC O:17.0/4 NXB XIC B29:6/11 BND OTE B22:10/3 NXB XIO B29:4/12 BST XIC O:17.0/4 NXB XIC B29:6/11 BND OTE B22:10/4 NXB BST BST XIO B29:4/13 NXB XIC B22:10/5 BND XIC B30:0/8 NXB XIC T21:17/DN XIO B29:4/13 BND OTE B22:10/5 NXB XIO B29:4/14 BST XIC O:17.0/4 NXB XIC B29:6/11 BND OTE B22:10/6 NXB XIO B29:4/15 OTE B22:10/7 NXB XIO B29:5/0 OTE B22:10/8 NXB BST XIC B29:4/13 NXB XIC B30:0/8 BND BST XIC O:17.0/4 NXB XIC B29:6/11 BND OTE B30:0/8 BND EOR
% Rung: 124 %
SOR XIC N9:1/7 BST XIC O:17.0/4 NXB XIC B29:6/11 BND XIO B29:4/13 XIO N7:20/3 TON T21:17 0.01 1000 0 EOR
% Rung: 125 %
SOR BST XIC B22:10/1 NXB XIC B22:10/2 NXB XIC B22:10/3 NXB XIC B22:10/4 NXB XIC B22:10/5 NXB XIC B22:10/6 NXB XIC B22:10/7 NXB XIC B22:10/8 BND XIO N7:20/1 OTE B22:4/2 EOR

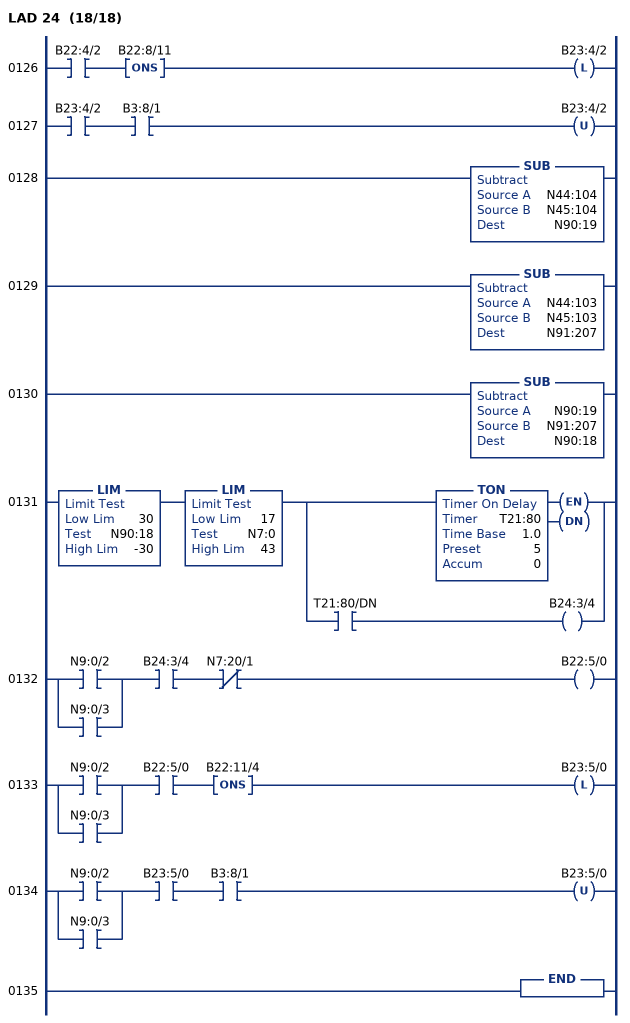
% Rung: 126 %
SOR XIC B22:4/2 OSR B22:8/11 OTL B23:4/2 EOR
% Rung: 127 %
SOR XIC B23:4/2 XIC B3:8/1 OTU B23:4/2 EOR
% Rung: 128 %
SOR SUB N44:104 N45:104 N90:19 EOR
% Rung: 129 %
SOR SUB N44:103 N45:103 N91:207 EOR
% Rung: 130 %
SOR SUB N90:19 N91:207 N90:18 EOR
% Rung: 131 %
SOR LIM 30 N90:18 -30 LIM 17 N7:0 43 BST TON T21:80 1.0 5 0 NXB XIC T21:80/DN OTE B24:3/4 BND EOR
% Rung: 132 %
SOR BST XIC N9:0/2 NXB XIC N9:0/3 BND XIC B24:3/4 XIO N7:20/1 OTE B22:5/0 EOR
% Rung: 133 %
SOR BST XIC N9:0/2 NXB XIC N9:0/3 BND XIC B22:5/0 OSR B22:11/4 OTL B23:5/0 EOR
% Rung: 134 %
SOR BST XIC N9:0/2 NXB XIC N9:0/3 BND XIC B23:5/0 XIC B3:8/1 OTU B23:5/0 EOR
% Rung: 135 %
SOR END EOR

LADDER 26
